PROGRAM P_Filtering
VAR
	//fbControlBlock : c_FB_ControlBlockWithMonito;
	fbFilterPa : FB_Filtering;
	fbFilterPb : FB_Filtering;
	fbFilterPs : FB_Filtering;
	fbFilterU : FB_Filtering;
	fbFilterPaLower : FB_Filtering;
END_VAR

fbFilterPa(
	ssMethodType := 1,
	Signal := G_OPC.fPa,
	Num := G_Parameter.fPressureFilterNum,
	Denz := G_Parameter.fPressureFilterDenz,
	Den := G_Parameter.fPressureFilterDen,
	Initial := G_Parameter.fPressureFilterInit,
	
	Signal_Filtered => G_Filtered.fPressurePistonSideFiltered,
	Signal_Filtered => G_OPC.fPaFiltered
);

fbFilterPb(
	ssMethodType := 1,
	Signal := G_OPC.fPb,
	Num := G_Parameter.fPressureFilterNum,
	Denz := G_Parameter.fPressureFilterDenz,
	Den := G_Parameter.fPressureFilterDen,
	Initial := G_Parameter.fPressureFilterInit,
	
	Signal_Filtered => G_Filtered.fPressureRodSideFiltered,
	Signal_Filtered => G_OPC.fPbFiltered
);

fbFilterPs(
	ssMethodType := 1,
	Signal := G_OPC.fPs,
	Num := G_Parameter.fPressureFilterNum,
	Denz := G_Parameter.fPressureFilterDenz,
	Den := G_Parameter.fPressureFilterDen,
	Initial := G_Parameter.fPressureFilterInit,
	
	Signal_Filtered => G_Filtered.fPressureSupplyFiltered,
	Signal_Filtered => G_OPC.fPsFiltered
);

fbFilterPaLower(
	ssMethodType := 1,
	Signal := G_OPC.fPaLower,
	Num := G_Parameter.fPressureFilterNum,
	Denz := G_Parameter.fPressureFilterDenz,
	Den := G_Parameter.fPressureFilterDen,
	Initial := G_Parameter.fPressureFilterInit,
	
	Signal_Filtered => G_Filtered.fPressureSupplyFiltered,
	Signal_Filtered => G_OPC.fPaLowerFiltered
);

//fbFilterU(
//	ssMethodType := 1,
//	Signal := G_Filtered.fValveOutputUnfiltered,
//	Num := G_Parameter.fSignalFilterNum,
//	Denz := G_Parameter.fSignalFilterDenz,
//	Den := G_Parameter.fSignalFilterDen,
//	Initial := G_Parameter.fSignalFilterInit,
//	
//	Signal_Filtered => G_Filtered.fValveOutputFiltered,
//	Signal_Filtered => G_OPC_UA.fFilteredSignal
//);

END_PROGRAM

(* stored: Version 1.1.0.1, ProductVersion 3.1.4024.12
   POU P_Filtering: Id {152e0fb1-83f0-480e-9255-787d93a44be7}, SpecialFunc None *)
